Universal Robots URScript: pick_up_bottle_cups_xijun.script

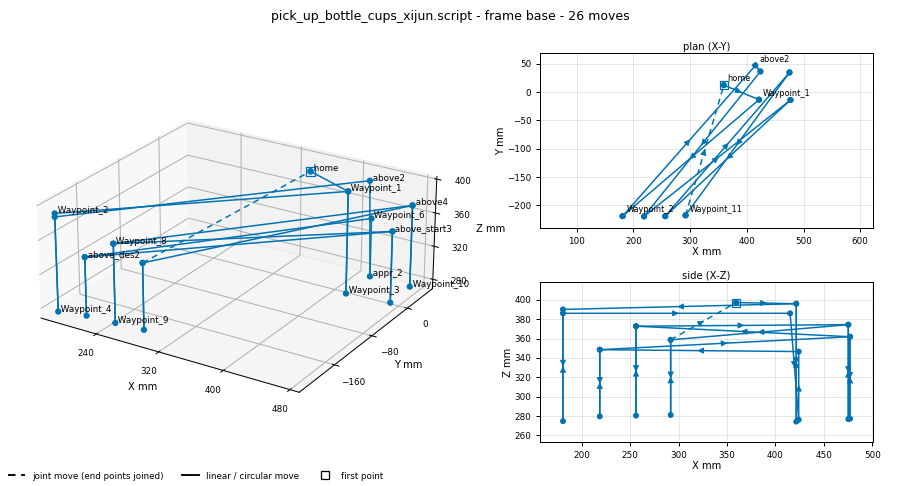
[picture p0: tool path of pick_up_bottle_cups_xijun.script in frame base, 26 of 27 moves have a stored position in this frame; points joined in program order, loops and branches not executed]
def pick_up_bottle_cups_xijun():
  set_tool_communication(True, 1000000, 2, 1, 1.5, 3.5)
  set_tool_output_mode(0)
  set_tool_digital_output_mode(0, 1)
  set_tool_digital_output_mode(1, 1)
  set_tool_voltage(24)
  set_tcp(p[0.0,0.0,0.0,0.0,0.0,0.0])
  set_target_payload(1.070000, [0.002000, 0.003000, 0.057000], [0.001723, 0.001723, 0.001723, 0.000000, 0.000000, 0.000000])
  set_safety_mode_transition_hardness(1)
  set_standard_analog_input_domain(0, 1)
  set_standard_analog_input_domain(1, 1)
  set_tool_analog_input_domain(0, 1)
  set_tool_analog_input_domain(1, 1)
  set_analog_outputdomain(0, 0)
  set_analog_outputdomain(1, 0)
  set_input_actions_to_default()
  step_count_40e01536_ad7e_4052_bcf8_2e85b5cb6fec = 0.0
  thread Step_Counter_Thread_e9fd1985_c531_4e2b_8333_d58f243b9e86():
    while (True):
      step_count_40e01536_ad7e_4052_bcf8_2e85b5cb6fec = step_count_40e01536_ad7e_4052_bcf8_2e85b5cb6fec + 1.0
      sync()
    end
  end
  run Step_Counter_Thread_e9fd1985_c531_4e2b_8333_d58f243b9e86()
  set_gravity([0.0, 0.0, 9.82])
  global Pallet_3_cnt=1
  global Plane_1=p[-0.700006141123905,1.3454883874109249E-6,0.3910559577028425,-1.2089868272251132,-1.2089999932245832,1.20858562628424]
  global Plane_2=p[0.0,0.0,0.0,0.0,0.0,0.0]
  global Point_1=p[0.6913645118948067,-0.12399382748223003,0.49223711947071,-1.2983729986843258,1.1259514972191385,-1.2203503861141718]
  # begin: URCap Installation Node
  #   Source: External Control, 1.0.5, FZI Research Center for Information Technology
  #   Type: External Control
  # end: URCap Installation Node
  # begin: URCap Installation Node
  #   Source: OnRobot, 6.2.0, OnRobot A/S
  #   Type: OnRobot Setup
  sleep(1)
  if (False):
    global rg_Busy = 0
    global rg_Depth = 0
    global rg_DepthRel = 0
    global rg_Grip_detected = 0
    global rg_Width = 0
  end
  ON_CONN_SHIFT_BOOL = 64
  ON_CONN_SHIFT_INT = 24
  ON_CONN_SHIFT_FLOAT = 24
  ON_CONN_REG_SUM_BOOL = 7
  ON_CONN_REG_SUM_INT = 4
  ON_CONN_REG_SUM_FLOAT = 3
  ON_TOOL_SHIFT_BOOL = 64
  ON_TOOL_SHIFT_INT = 25
  ON_TOOL_SHIFT_FLOAT = 24
  ON_TOOL_SHIFT_BOOL_ARR = [64, 71, 71]
  ON_TOOL_SHIFT_INT_ARR = [25, 28, 28]
  ON_TOOL_SHIFT_FLOAT_ARR = [24, 27, 27]
  ON_TOOL_REG_SUM_BOOL = 7
  ON_TOOL_REG_SUM_INT = 3
  ON_TOOL_REG_SUM_FLOAT = 3
  ON_REGISTERS_SPEEDL_FLOAT = 0
  ON_REG_USE_TOOL = False
  ON_DI_SINGLE = 0
  ON_DI_PRIMARY = 1
  ON_DI_SECONDARY = 2
  ON_DI_DUAL = 3
  on_robot_type = 10
  on_robot_cycle = 2.0
  on_conn_ip = "localhost"
  on_tool_ip = "localhost"
  on_device_socket_port = 51234
  on_conn_xmlrpc = rpc_factory("xmlrpc", "http://localhost:41414")
  on_tool_xmlrpc = rpc_factory("xmlrpc", "http://localhost:41414")
  on_RPC = rpc_factory("xmlrpc", "http://127.0.0.1:31416")
  ON_DEBUG_LOG = False
  on_isMetric = True
  on_toolConnector = True
  on_ioqc = False
  on_dual = False
  on_computebox = False
  on_devices = 1
  on_gripper = [False, False, False]
  on_custom_tcp_id = "none"
  on_custom_tcp_enabled = False
  speedlTime = 0.001
  on_ft = False
  rg_index = 0
  on_gripper[rg_index] = True
  #======    OnRobot Globals    ======#

  ON_MATH_PI=3.141593
  ON_ZEROPOSE=p[0.0,0.0,0.0,0.0,0.0,0.0]
  ON_ZEROFRAME=p[0.0,0.0,0.0,0.0,0.0,0.0]
  ON_ZERO3D=[0.0,0.0,0.0]
  ON_ZERO6D=[0.0,0.0,0.0,0.0,0.0,0.0]
  ON_ZERO8D=[0.0,0.0,0.0,0.0,0.0,0.0,0.0,0.0]
  ON_FALSE3D=[False,False,False]
  ON_FALSE6D=[False,False,False,False,False,False]
  ON_FALSE8D=[False,False,False,False,False,False,False,False]
  global on_return=0
  on_speedL=ON_ZERO6D
  on_speedBase=ON_ZERO6D
  on_speedVect=ON_ZERO6D
  on_speedExtra=ON_ZERO6D
  on_speedCB=ON_ZERO6D
  on_speedGecko=ON_ZERO6D
  on_RTDE_error=0
  on_RTDE_tool_error=0
  on_dataProcess_thrd=0
  ON_DEVICE_ID_MISSING=0
  ON_INIT_WATCHDOG_HZ=5
  ON_INIT_TIMEOUT=2000
  on_robot_TCP_offset=ON_ZEROFRAME
  on_tcp_offset_actual=ON_ZEROFRAME
  on_cog_actual=ON_ZEROFRAME
  on_mass_actual=0.0
  on_robot_mount=[0.0,0.0]

  #======    End of OnRobot Globals    ======#
  #======    OnRobot RG Globals    ======#

  RG_DEVICE_ID_RG2=32
  RG_DEVICE_ID_RG6=33
  if ON_DEBUG_LOG:
  textmsg("RG Dual: False, Index: ",rg_index)
  if False:
  rg_index=-1
  end
  end
  rg_Width_arr=[0,0,0]
  rg_Depth_arr=[0,0,0]
  rg_DepthRel_arr=[0,0,0]
  rg_product_code_arr=[0,0,0]
  rg_device_id_arr=[0,0,0]
  rg_Status_arr=[0,0,0]
  rg_Grip_detected_arr=[False,False,False]
  rg_Busy_arr=[False,False,False]
  rg_S1_pushed_arr=[False,False,False]
  rg_S1_triggered_arr=[False,False,False]
  rg_S2_pushed_arr=[False,False,False]
  rg_S2_triggered_arr=[False,False,False]
  rg_Safety_error_arr=[False,False,False]
  rg_Speed_arr=[0,0,0]
  rg_Angle_arr=[0,0,0]
  rg_Angle_speed_arr=[0,0,0]
  rg_Depth_prev_arr=[0,0,0]
  rg_speedDC=ON_ZERO6D
  rg_data_error_arr=[0,0,0]
  rg_mounting_angle_arr=[0,0,0]
  rg_fingertip_arr=[0,0,0]
  rg_Grip_guard_arr=[False,False,False]

  rg_Width=0
  rg_Depth=0
  rg_DepthRel=0
  rg_Busy=False
  rg_Grip_detected=False
  def get_rg_Width():
  return rg_Width
  end
  def get_rg_Depth():
  return rg_Depth
  end
  def get_rg_DepthRel():
  return rg_DepthRel
  end
  def get_rg_Busy():
  return rg_Busy
  end
  def get_rg_Grip_detected():
  return rg_Grip_detected
  end

  rg2_mount_bracket_offset=35.0/1000.0
  rg2_mount_body_offset=p[0.0,0.0,0.180,0.0,0.0,0.0]
  rg2_mount_cog_offset=p[0.0,0.0,0.065,0.0,0.0,0.0]
  rg6_mount_bracket_offset=35.0/1000.0
  rg6_mount_body_offset=p[0.0,0.0,0.230,0.0,0.0,0.0]
  rg6_mount_cog_offset=p[0.0,0.0,0.080,0.0,0.0,0.0]

  #======    End of OnRobot RG Globals    ======#
  #======    OnRobot Interface Messages    ======#

  on_devices_primary_log="OnRobot Devices"
  on_devices_secondary_log="OnRobot Secondary Device"
  on_program_halted="<br>Program halted."
  on_device_error_title="OnRobot - Device error"
  on_install_error="OnRobot Setup is not correct.<br>Check the status in the OnRobot Setup page in the Installation Tab.<br>Program halted."
  on_device_missing="No device connected.<br>Program halted."
  cb_device_missing="No OnRobot Compute Box connected.<br>Program halted."
  ft_device_missing="No OnRobot FT sensor or license detected.<br>Program halted."
  hex_device_missing="No HEX sensor connected.<br>Program halted."
  rg2ft_device_missing="No RG2-FT gripper connected.<br>Program halted."
  rg_device_missing="No RG gripper connected.<br>Program halted."
  vg_device_missing="No VG gripper connected.<br>Program halted."
  gg_device_missing="No Gecko Gripper connected.<br>Program halted."
  sg_device_missing="No Soft Gripper connected.<br>Program halted."
  tfg_device_missing="No 3FG gripper connected.<br>Program halted."
  sdr_device_missing="No OnRobot Sander connected.<br>Program halted."
  twofg_device_missing="No 2FG gripper connected.<br>Program halted."
  vgp_device_missing="No VGP gripper connected.<br>Program halted."
  mg_device_missing="No Magnetic Gripper connected.<br>Program halted."
  fgp_device_missing="No 2FGP20 Gripper connected.<br>Program halted."
  eyes_device_missing="No OnRobot Eyes connected.<br>Program halted."
  on_xmlrpc_start_ip="Connecting to OnRobot XML-RPC Server:"
  on_java_comm_error_textmsg_title="OnRobot - Communication error:"
  on_java_comm_controlsocket_open_error="Socket 'javaSocket' opening was unsuccessful."
  on_java_comm_error_title="OnRobot - Communication error"
  on_java_comm_socket_open_error="Establishing connection with the URCap was timed out.<br>Check the status in the OnRobot Setup page in the Installation Tab.<br>Program halted."
  on_rtde_feed_error_textmsg_title="OnRobot - RTDE error:"
  on_rtde_feed_error="RTDE feed error. OnRobot device count mismatch.<br>Program halted."
  on_rtde_feed_tool_error="Tool RTDE feed error. OnRobot device count mismatch.<br>Program halted."
  on_rtde_feed_open_error_textmsg="Socket 'rtdeFeed' opening was unsuccessful."
  on_rtde_feed_error_title="OnRobot - RTDE error"
  on_rtde_feed_count_error="Invalid RTDE offset setup detected. Please check RTDE Offsets at the OnRobot Setup page in the Installation Tab.<br>Program halted."
  on_rtde_feed_open_error="Establishing connection with the devices was timed out.<br>Ensure that the OnRobot devices are operational, and check the status in the OnRobot Setup page in the Installation Tab."

  #======    End of OnRobot Interface Messages    ======#
  #======    OnRobot Interface    ======#

  on_portopened_javaSocket=False
  on_rtde_feed_opened=False
  on_dataProcess_running=False
  def on_missing():
  popup(on_device_missing,title=on_device_error_title,error=True,blocking=False)
  halt
  end
  def cb_missing():
  popup(cb_device_missing,title=on_device_error_title,error=True,blocking=False)
  halt
  end
  def ft_missing():
  popup(ft_device_missing,title=on_device_error_title,error=True,blocking=False)
  halt
  end
  def hex_missing():
  popup(hex_device_missing,title=on_device_error_title,error=True,blocking=False)
  halt
  end
  def rg2ft_missing():
  popup(rg2ft_device_missing,title=on_device_error_title,error=True,blocking=False)
  halt
  end
  def rg_missing():
  popup(rg_device_missing,title=on_device_error_title,error=True,blocking=False)
  halt
  end
  def vg_missing():
  popup(vg_device_missing,title=on_device_error_title,error=True,blocking=False)
  halt
  end
  def gg_missing():
  popup(gg_device_missing,title=on_device_error_title,error=True,blocking=False)
  halt
  end
  def sg_missing():
  popup(sg_device_missing,title=on_device_error_title,error=True,blocking=False)
  halt
  end
  def tfg_missing():
  popup(tfg_device_missing,title=on_device_error_title,error=True,blocking=False)
  halt
  end
  def sdr_missing():
  popup(sdr_device_missing,title=on_device_error_title,error=True,blocking=False)
  halt
  end
  def twofg_missing():
  popup(twofg_device_missing,title=on_device_error_title,error=True,blocking=False)
  halt
  end
  def vgp_missing():
  popup(vgp_device_missing,title=on_device_error_title,error=True,blocking=False)
  halt
  end
  def mg_missing():
  popup(mg_device_missing,title=on_device_error_title,error=True,blocking=False)
  halt
  end
  def fgp_missing():
  popup(fgp_device_missing,title=on_device_error_title,error=True,blocking=False)
  halt
  end
  def eyes_missing():
  popup(eyes_device_missing,title=on_device_error_title,error=True,blocking=False)
  halt
  end
  def on_portclose_javaSocket():
  socket_close("javaSocket")
  on_portopened_javaSocket=False
  end
  def on_portopen_javaSocket():
  on_portclose_javaSocket()
  on_portopened_javaSocket=socket_open("127.0.0.1",44005,"javaSocket")
  if not on_portopened_javaSocket:
  textmsg(on_java_comm_error_textmsg_title,on_java_comm_controlsocket_open_error)
  popup(on_java_comm_socket_open_error,title=on_java_comm_error_title,error=True,blocking=False)
  halt
  end
  end
  on_conn_rtde_feed_name="rtdeFeedConn"
  on_tool_rtde_feed_name="rtdeFeedTool"
  def on_rtde_feed_close(rtdeFeedName):
  socket_close(rtdeFeedName)
  on_rtde_feed_opened=False
  end
  def on_rtde_feed_open(deviceIP,rtdeFeedName,regStart,regSum,regSpeedl):
  on_rtde_feed_close(rtdeFeedName)
  if((regStart[0]+regSum[0])>128)or((regStart[1]+regSum[1])>48)or((regStart[2]+regSum[2])>48):
  popup(on_rtde_feed_count_error,title=on_rtde_feed_error_title,error=True,blocking=False)
  textmsg(str_cat("RegStart: ",regStart),str_cat("  -  RegSum: ",regSum))
  halt
  end
  on_rtde_feed_opened=socket_open(deviceIP,on_device_socket_port,rtdeFeedName)
  if not on_rtde_feed_opened:
  on_rtde_feed_opened=socket_open(deviceIP,on_device_socket_port,rtdeFeedName)
  end
  if not on_rtde_feed_opened:
  textmsg(on_rtde_feed_error_textmsg_title,on_rtde_feed_open_error_textmsg)
  popup(on_rtde_feed_open_error,title=on_rtde_feed_error_title,error=True,blocking=False)
  halt
  end
  socket_send_int(regStart[0],rtdeFeedName)
  socket_send_int(regSum[0],rtdeFeedName)
  socket_send_int(regStart[1],rtdeFeedName)
  socket_send_int(regSum[1],rtdeFeedName)
  socket_send_int(regStart[2],rtdeFeedName)
  socket_send_int(regSum[2],rtdeFeedName)
  socket_send_int(regSpeedl,rtdeFeedName)
  socket_send_int(on_devices,rtdeFeedName)
  end
  def on_dataRead():
  enter_critical
  on_RTDE_error=read_input_integer_register(ON_CONN_SHIFT_INT)
  if(ON_REG_USE_TOOL):
  on_RTDE_tool_error=read_input_integer_register(ON_TOOL_SHIFT_INT_ARR[0])
  end
  exit_critical
  end
  def on_set_rtde_watchdog(updateHz=ON_INIT_WATCHDOG_HZ):
  local effect="stop"
  if(updateHz<1):
  effect="ignore"
  end
  watchdog_conn_reg_str=str_cat("input_int_register_",ON_CONN_SHIFT_INT)
  rtde_set_watchdog(watchdog_conn_reg_str,updateHz,effect)
  if(ON_REG_USE_TOOL):
  watchdog_tool_reg_str=str_cat("input_int_register_",ON_TOOL_SHIFT_INT_ARR[0])
  rtde_set_watchdog(watchdog_tool_reg_str,updateHz,effect)
  end
  if ON_DEBUG_LOG:
  local update_str=str_cat(" "+effect+" watchdog set to [Hz]: ",updateHz)
  textmsg(watchdog_conn_reg_str,update_str)
  if(ON_REG_USE_TOOL):
  local update_str=str_cat(" "+effect+" watchdog set to [Hz]: ",updateHz)
  textmsg(watchdog_tool_reg_str,update_str)
  end
  end
  end
  def on_speedCB_get():
  return[on_speedCB[0],on_speedCB[1],on_speedCB[2],on_speedCB[3],on_speedCB[4],on_speedCB[5]]
  end
  def on_speedGecko_get():
  local speedExtra=ON_ZERO6D
  if on_speedl_for_gecko:
  speedExtra=[on_speedGecko[0],on_speedGecko[1],on_speedGecko[2],on_speedGecko[3],on_speedGecko[4],on_speedGecko[5]]
  end
  return speedExtra
  end
  def on_speedGecko_set(speedGecko):
  on_speedGecko=[speedGecko[0],speedGecko[1],speedGecko[2],speedGecko[3],speedGecko[4],speedGecko[5]]
  end
  thread on_dataProcess_thread():
  if ON_DEBUG_LOG:
  textmsg("Starting on_dataRead thread")
  end
  local error=False
  on_dataProcess_running=True
  sync()
  while on_dataProcess_running:
  sync()
  on_dataRead()
  error=on_error((on_RTDE_error<0),on_rtde_feed_error,on_rtde_feed_error_title,error)
  error=on_error((ON_REG_USE_TOOL and(on_RTDE_tool_error<0)),on_rtde_feed_tool_error,on_rtde_feed_error_title,error)
  on_dataProcess_running=not error
  end
  if error:
  halt
  end
  if ON_DEBUG_LOG:
  textmsg("Stopping on_dataRead thread")
  end
  end
  thread on_set_watchdog_thread():
  sleep(2)
  on_set_rtde_watchdog(updateHz=ON_INIT_WATCHDOG_HZ)
  sleep(1/ON_INIT_WATCHDOG_HZ)
  on_dataProcess_running=False
  kill on_dataProcess_thrd
  end

  #======    End of OnRobot Interface    ======#
  #======    OnRobot QC Setup Tool Connector    ======#

  def tc_setup_tool():
  if ON_DEBUG_LOG:
  textmsg("QC Setup Tool Connector start...")
  end
  set_tool_voltage(24)

  set_tool_communication(True,1000000,2,1,1.5,3.5)

  if ON_DEBUG_LOG:
  textmsg("QC Setup Tool Connector end.")
  end
  end

  #======    End of OnRobot QC Setup Tool Connector    ======#
  #======    OnRobot RG Interface    ======#

  rg_dataRead_running=False
  def rg_dataRead_RTDE(tool_index):
  local reg_offset_bool=ON_TOOL_SHIFT_BOOL_ARR[tool_index]
  local reg_offset_int=ON_TOOL_SHIFT_INT_ARR[tool_index]
  local reg_offset_float=ON_TOOL_SHIFT_FLOAT_ARR[tool_index]
  enter_critical
  floatRegDummy=read_input_float_register(reg_offset_float+0)
  rg_Width_arr[tool_index]=floatRegDummy
  floatRegDummy=read_input_float_register(reg_offset_float+1)
  rg_Depth_arr[tool_index]=floatRegDummy
  floatRegDummy=read_input_float_register(reg_offset_float+2)
  rg_DepthRel_arr[tool_index]=floatRegDummy
  intRegDummy=read_input_integer_register(reg_offset_int+0)
  rg_device_id_arr[tool_index]=intRegDummy
  intRegDummy=read_input_integer_register(reg_offset_int+1)
  rg_product_code_arr[tool_index]=intRegDummy
  intRegDummy=read_input_integer_register(reg_offset_int+2)
  rg_Status_arr[tool_index]=intRegDummy
  boolRegDummy=read_input_boolean_register(reg_offset_bool+0)
  rg_Busy_arr[tool_index]=boolRegDummy
  boolRegDummy=read_input_boolean_register(reg_offset_bool+1)
  rg_Grip_detected_arr[tool_index]=boolRegDummy
  boolRegDummy=read_input_boolean_register(reg_offset_bool+2)
  rg_S1_pushed_arr[tool_index]=boolRegDummy
  boolRegDummy=read_input_boolean_register(reg_offset_bool+3)
  rg_S1_triggered_arr[tool_index]=boolRegDummy
  boolRegDummy=read_input_boolean_register(reg_offset_bool+4)
  rg_S2_pushed_arr[tool_index]=boolRegDummy
  boolRegDummy=read_input_boolean_register(reg_offset_bool+5)
  rg_S2_triggered_arr[tool_index]=boolRegDummy
  boolRegDummy=read_input_boolean_register(reg_offset_bool+6)
  rg_Safety_error_arr[tool_index]=boolRegDummy
  exit_critical
  end
  thread rg_dataRead_thread():
  if ON_DEBUG_LOG:
  textmsg("Starting rg_dataRead thread")
  end
  while rg_dataRead_running:
  sync()
  rg_Depth_prev_arr=rg_Depth_arr
  if(rg_index==ON_DI_DUAL):
  rg_dataRead_RTDE(ON_DI_PRIMARY)
  rg_dataRead_RTDE(ON_DI_SECONDARY)
  else:
  rg_dataRead_RTDE(rg_index)
  end
  end
  if ON_DEBUG_LOG:
  textmsg("Stopping rg_dataRead thread")
  end
  end

  #======    End of OnRobot RG Interface    ======#
  #======    OnRobot TCP Messages    ======#

  on_tcp_log_msg_default="OnRobot: Robot TCP Offset set to:"
  on_tcp_log_msg_primary="OnRobot: Robot TCP Offset set to Primary:"
  on_tcp_log_msg_secondary="OnRobot: Robot TCP Offset set to Secondary:"

  #======    End of OnRobot TCP Messages    ======#
  #======    OnRobot TCP    ======#

  on_tcp_offset_actual=ON_ZEROFRAME
  on_tcp_offset_primary=ON_ZEROFRAME
  on_tcp_static_primary=ON_ZEROFRAME
  on_tcp_dynamic_primary=ON_ZEROFRAME
  on_tcp_adapters=ON_ZEROFRAME
  on_tcp_qc_primary=ON_ZEROFRAME
  on_tcp_base_primary=ON_ZEROFRAME
  on_tcp_gripper_static_primary=ON_ZEROFRAME
  on_tcp_workpiece_primary=ON_ZEROFRAME
  on_tcp_gripper_dynamic_primary=ON_ZEROFRAME
  on_tcp_gripper_primary=ON_ZEROFRAME
  on_tcp_offset_secondary=ON_ZEROFRAME
  on_tcp_static_secondary=ON_ZEROFRAME
  on_tcp_dynamic_secondary=ON_ZEROFRAME
  on_tcp_qc_secondary=ON_ZEROFRAME
  on_tcp_base_secondary=ON_ZEROFRAME
  on_tcp_gripper_static_secondary=ON_ZEROFRAME
  on_tcp_workpiece_secondary=ON_ZEROFRAME
  on_tcp_gripper_dynamic_secondary=ON_ZEROFRAME
  on_tcp_gripper_secondary=ON_ZEROFRAME
  on_tcp_custom_preset_assigned=False
  on_tcp_custom_preset=ON_ZEROFRAME
  def on_tcp_init_adapters():
  if ON_DEBUG_LOG:
  textmsg("TCP Init Adapters start..")
  end
  enter_critical
  on_tcp_adapters=ON_ZEROFRAME
  local adapterCount=length(on_tcp_adapters_array)
  local i=0
  while(i<adapterCount):
  on_tcp_adapters=pose_trans(on_tcp_adapters,on_tcp_adapters_array[i])
  i=i+1
  end
  exit_critical
  if ON_DEBUG_LOG:
  textmsg("TCP Init Adapters end.")
  end
  end
  def on_tcp_update_primary():
  if ON_DEBUG_LOG:
  textmsg("TCP Update Primary start..")
  end
  on_tcp_gripper_dynamic_primary=p[0.0, 0.0, 0.0, 0.0, 0.0, 0.0]
  enter_critical
  on_tcp_dynamic_primary=pose_trans(on_tcp_static_primary,on_tcp_gripper_dynamic_primary)
  on_tcp_offset_primary=pose_trans(on_tcp_dynamic_primary,on_tcp_workpiece_primary)
  exit_critical
  if ON_DEBUG_LOG:
  textmsg("TCP Update Primary end.")
  end
  end
  def on_tcp_init_primary():
  if ON_DEBUG_LOG:
  textmsg("TCP Init Primary start..")
  end
  enter_critical
  on_tcp_base_primary=pose_trans(on_tcp_adapters,on_tcp_qc_primary)
  on_tcp_static_primary=pose_trans(on_tcp_base_primary,on_tcp_gripper_static_primary)
  exit_critical
  on_tcp_update_primary()
  if ON_DEBUG_LOG:
  textmsg("TCP Init Primary end.")
  end
  end
  def on_tcp_offset_set(TCP_offset):
  if ON_DEBUG_LOG:
  textmsg("TCP Offset set started!")
  end
  on_tcp_offset_send(TCP_offset)
  if(on_follow_tcp):
  set_tcp(TCP_offset)
  end
  on_robot_TCP_offset=TCP_offset
  if ON_DEBUG_LOG:
  textmsg("TCP Offset set to: ",on_robot_TCP_offset)
  end
  end
  def on_tcp_offset_forced_set_actual(isPrimary=True):
  if(not on_follow_tcp):

  local tcp_log_msg=on_tcp_log_msg_default

  textmsg(tcp_log_msg,on_tcp_offset_actual)
  set_tcp(on_tcp_offset_actual)
  end
  end
  def on_tcp_update(isPrimary=True):
  on_tcp_update_primary()

  on_tcp_set_actual_to(isPrimary)
  end
  def on_tcp_set_actual_to(isPrimary=True):

  on_tcp_offset_actual=on_tcp_offset_primary
  if(on_follow_tcp):
  textmsg(on_tcp_log_msg_default,on_tcp_offset_actual)
  end

  on_tcp_active_is_primary=isPrimary
  on_tcp_offset_set(on_tcp_offset_actual)
  end
  def on_tcp_update_workpiece_primary(workpiece_offset):
  if ON_DEBUG_LOG:
  textmsg("TCP Update Tool Primary start..")
  end
  on_tcp_workpiece_primary=workpiece_offset
  on_tcp_update_primary()
  if ON_DEBUG_LOG:
  textmsg("TCP Update Tool Primary end.")
  end
  end
  def on_tcp_workpiece_rpy_get(xyz=[0.0,0.0,0.0],rpy=[0.0,0.0,0.0]):
  local rotvec=rpy2rotvec(rpy)
  local workpiece_offset=p[xyz[0],xyz[1],xyz[2],rotvec[0],rotvec[1],rotvec[2]]
  return workpiece_offset
  end

  def on_tcp_update_workpiece(workpiece_offset,tool_index=0):
  if ON_DEBUG_LOG:
  textmsg("TCP Update Tool start..")
  end
  if(tool_index!=ON_DI_SECONDARY):
  on_tcp_update_workpiece_primary(workpiece_offset)
  local isPrimary=True

  end
  on_tcp_set_actual_to(isPrimary)
  if ON_DEBUG_LOG:
  textmsg("TCP Update Tool end.")
  end
  end
  def on_get_tcp_for(tool_index):
  if tool_index==ON_DI_SECONDARY:
  local actual_tcp=on_tcp_static_secondary
  else:
  local actual_tcp=on_tcp_static_primary
  end
  return actual_tcp
  end
  def on_tcp_custom_unused():
  return ON_ZEROFRAME
  end
  def on_tcp_update_custom():
  if ON_DEBUG_LOG:
  textmsg("TCP Update Custom start..")
  end
  if(on_custom_tcp_enabled):
  on_tcp_custom_unused()
  on_tcp_custom_unused()
  on_tcp_custom_unused()
  on_tcp_custom_unused()

  end
  if ON_DEBUG_LOG:
  textmsg("TCP Update Custom end.")
  end
  end

  #======    End of OnRobot TCP    ======#
  #======    OnRobot Payload Messages    ======#

  on_mass_log_msg="OnRobot: Robot Payload Mass set to:"
  on_cog_log_msg="OnRobot: Robot Payload Center of Gravity set to:"

  #======    End of OnRobot Payload Messages    ======#
  #======    OnRobot Payload    ======#

  on_cog_actual=ON_ZEROFRAME
  on_mass_actual=0.0
  on_cog_primary=ON_ZEROFRAME
  on_cog_L1L2_primary=ON_ZEROFRAME
  on_mass_primary=0.0
  on_mass_L1L2_primary=0.0
  on_cog_adapters=ON_ZEROFRAME
  on_cog_qc_primary=ON_ZEROFRAME
  on_cog_base_primary=ON_ZEROFRAME
  on_cog_gripper_primary=ON_ZEROFRAME
  on_cog_workpiece_primary=ON_ZEROFRAME
  on_mass_adapters=0.0
  on_mass_qc_primary=0.0
  on_mass_base_primary=0.0
  on_mass_gripper_primary=0.0
  on_mass_workpiece_primary=0.0
  on_cog_secondary=ON_ZEROFRAME
  on_mass_secondary=0.0
  on_cog_gripper_secondary=ON_ZEROFRAME
  on_mass_gripper_secondary=0.0
  on_cog_workpiece_secondary=ON_ZEROFRAME
  on_mass_workpiece_secondary=0.0
  ON_LB2KG001=0.45359237/100
  def on_payload_init_adapters():
  if ON_DEBUG_LOG:
  textmsg("TCP Init Adapters start..")
  end
  enter_critical
  on_cog_adapters=ON_ZEROFRAME
  on_mass_adapters=0.0
  local massLAL0Ratio=0
  local adapterAbsCOG=ON_ZEROFRAME
  local tcp_adapter_offset=ON_ZEROFRAME
  local adapterCount=length(on_tcp_adapters_array)
  local i=0
  while(i<adapterCount):
  on_mass_adapters=on_mass_adapters+on_mass_adapters_array[i]
  if(on_mass_adapters<=0):
  massLAL0Ratio=0
  else:
  massLAL0Ratio=on_mass_adapters_array[i]/on_mass_adapters
  end
  adapterAbsCOG=pose_trans(tcp_adapter_offset,on_tcp_adapters_array[i])
  adapterAbsCOG=p[adapterAbsCOG[0],adapterAbsCOG[1],adapterAbsCOG[2],0.0,0.0,0.0]
  on_cog_adapters=interpolate_pose(on_cog_adapters,adapterAbsCOG,massLAL0Ratio)
  on_cog_adapters=p[on_cog_adapters[0],on_cog_adapters[1],on_cog_adapters[2],0.0,0.0,0.0]
  tcp_adapter_offset=pose_trans(tcp_adapter_offset,on_tcp_adapters_array[i])
  i=i+1
  sync()
  end
  exit_critical
  if ON_DEBUG_LOG:
  textmsg("TCP Init Adapters end.")
  end
  end
  def on_payload_update_primary():
  if ON_DEBUG_LOG:
  textmsg("Payload Update Primary start..")
  end
  enter_critical
  on_mass_primary=on_mass_L1L2_primary+on_mass_workpiece_primary
  local massL1L2L3Ratio=on_mass_workpiece_primary/on_mass_primary
  local workpieceAbsCOG=pose_trans(on_tcp_dynamic_primary,on_cog_workpiece_primary)
  workpieceAbsCOG=p[workpieceAbsCOG[0],workpieceAbsCOG[1],workpieceAbsCOG[2],0.0,0.0,0.0]
  on_cog_primary=interpolate_pose(on_cog_L1L2_primary,workpieceAbsCOG,massL1L2L3Ratio)
  on_cog_primary=p[on_cog_primary[0],on_cog_primary[1],on_cog_primary[2],0.0,0.0,0.0]
  exit_critical
  if ON_DEBUG_LOG:
  textmsg("Payload Update Primary end.")
  end
  end
  def on_payload_init_primary():
  if ON_DEBUG_LOG:
  textmsg("Payload Init Primary start..")
  end
  enter_critical
  on_mass_base_primary=on_mass_adapters+on_mass_qc_primary
  local massL0L1Ratio=on_mass_qc_primary/on_mass_base_primary
  on_mass_L1L2_primary=on_mass_base_primary+on_mass_gripper_primary
  local massL1L2Ratio=on_mass_gripper_primary/on_mass_L1L2_primary
  local qcAbsCOG=pose_trans(on_tcp_adapters,on_cog_qc_primary)
  qcAbsCOG=p[qcAbsCOG[0],qcAbsCOG[1],qcAbsCOG[2],0.0,0.0,0.0]
  on_cog_base_primary=interpolate_pose(on_cog_adapters,qcAbsCOG,massL0L1Ratio)
  on_cog_base_primary=p[on_cog_base_primary[0],on_cog_base_primary[1],on_cog_base_primary[2],0.0,0.0,0.0]
  local gripperAbsCOG=pose_trans(on_tcp_base_primary,on_cog_gripper_primary)
  gripperAbsCOG=p[gripperAbsCOG[0],gripperAbsCOG[1],gripperAbsCOG[2],0.0,0.0,0.0]
  on_cog_L1L2_primary=interpolate_pose(on_cog_base_primary,gripperAbsCOG,massL1L2Ratio)
  on_cog_L1L2_primary=p[on_cog_L1L2_primary[0],on_cog_L1L2_primary[1],on_cog_L1L2_primary[2],0.0,0.0,0.0]
  exit_critical
  on_payload_update_primary()
  if ON_DEBUG_LOG:
  textmsg("Payload Init Primary end.")
  end
  end
  def on_payload_update():
  on_payload_update_primary()

  on_mass_actual =on_mass_primary
  on_cog_actual=on_cog_primary

  on_payload_set_actual()
  end
  def on_payload_set_actual():

  on_mass_actual =on_mass_primary
  on_cog_actual=on_cog_primary

  local CoG=[on_cog_actual[0],on_cog_actual[1],on_cog_actual[2]]
  on_payload_set(on_mass_actual,CoG)
  end
  def on_payload_update_workpiece_primary(workpiece_mass=0,workpiece_cog=[0.0,0.0,0.0]):
  if ON_DEBUG_LOG:
  textmsg("Payload Update Workpiece Primary start..")
  end
  on_cog_workpiece_primary=p[workpiece_cog[0],workpiece_cog[1],workpiece_cog[2],0.0,0.0,0.0]
  on_mass_workpiece_primary=workpiece_mass
  on_payload_update_primary()
  if ON_DEBUG_LOG:
  textmsg("Payload Update Workpiece Primary end.")
  end
  end
  def on_payload_set(mass,CoG):
  if ON_DEBUG_LOG:
  textmsg("Payload set started!")
  end
  local center_of_gravity=[CoG[0],CoG[1],CoG[2]]
  on_payload_send(center_of_gravity,mass)
  if(on_isMetric):
  local roundedMass=floor(mass*100+0.5)/100
  else:
  local roundedMass=floor(mass/ON_LB2KG001+0.5)*ON_LB2KG001
  end
  set_payload(roundedMass,center_of_gravity)
  on_mass_actual=roundedMass
  on_cog_actual=p[CoG[0],CoG[1],CoG[2],0.0,0.0,0.0]
  if ON_DEBUG_LOG:
  textmsg("Payload mass, CoG set to: ",str_cat(str_cat(mass,", "),CoG))
  end
  end

  def on_payload_update_secondary():
  end
  def on_payload_init_secondary():
  end

  def on_payload_update_workpiece(workpiece_mass,workpiece_cog=[0.0,0.0,0.0],tool_index=0):
  if ON_DEBUG_LOG:
  textmsg("Payload Update Workpiece start..")
  end
  if(tool_index!=ON_DI_SECONDARY):
  on_cog_workpiece_primary=p[workpiece_cog[0],workpiece_cog[1],workpiece_cog[2],0.0,0.0,0.0]
  on_mass_workpiece_primary=workpiece_mass
  else:
  on_cog_workpiece_secondary=p[workpiece_cog[0],workpiece_cog[1],workpiece_cog[2],0.0,0.0,0.0]
  on_mass_workpiece_secondary=workpiece_mass
  end
  on_payload_update()
  if ON_DEBUG_LOG:
  textmsg("Payload Update Workpiece end.")
  end
  end
  def on_payload_get_cog2tcp_workpiece(tool_index=0):
  if(tool_index!=ON_DI_SECONDARY):
  local cog_tool=[on_tcp_workpiece_primary[0],on_tcp_workpiece_primary[1],on_tcp_workpiece_primary[2]]
  else:
  local cog_tool=[on_tcp_workpiece_secondary[0],on_tcp_workpiece_secondary[1],on_tcp_workpiece_secondary[2]]
  end
  return cog_tool
  end

  #======    End of OnRobot Payload    ======#
  #======    OnRobot QC TCP    ======#

  onrobotmini=0

  def on_tcp_offset_send(TCP_offset):
  on_robot_TCP_offset=TCP_offset
  end
  def on_payload_send(CoG,mass):
  on_robot_payload_cog=CoG
  on_robot_payload_mass=mass
  end


  #======    End of OnRobot QC TCP    ======#
  #======    OnRobot RG TCP    ======#

  def rg_mount_tcp(gripper_angle,isRG2=True):
  if ON_DEBUG_LOG:
  textmsg("RG Mount TCP command starting..")
  end
  if(isRG2):
  local gripperBracket=rg2_mount_bracket_offset
  local gripperBody=rg2_mount_body_offset
  else:
  local gripperBracket=rg6_mount_bracket_offset
  local gripperBody=rg6_mount_body_offset
  end
  local gripperRotVec=rpy2rotvec([gripper_angle,0.0,0.0])
  local gripperMountOffset=p[0.0,0.0,gripperBracket,gripperRotVec[0],gripperRotVec[1],gripperRotVec[2]]
  local gripperOffsetStatic=pose_trans(gripperMountOffset,gripperBody)
  if ON_DEBUG_LOG:
  textmsg("RG Mount TCP command ended.")
  end
  return gripperOffsetStatic
  end
  def rg_mount_cog(gripper_angle,isRG2=True):
  if ON_DEBUG_LOG:
  textmsg("RG Mount CoG command starting..")
  end
  if(isRG2):
  local gripperBracket=rg2_mount_bracket_offset
  local gripperCoG=rg2_mount_cog_offset
  else:
  local gripperBracket=rg6_mount_bracket_offset
  local gripperCoG=rg6_mount_cog_offset
  end
  local gripperRotVec=rpy2rotvec([gripper_angle,0.0,0.0])
  local gripperMountOffset=p[0.0,0.0,gripperBracket,gripperRotVec[0],gripperRotVec[1],gripperRotVec[2]]
  local gripperCOGOffset=pose_trans(gripperMountOffset,gripperCoG)
  gripperCOGOffset=p[gripperCOGOffset[0],gripperCOGOffset[1],gripperCOGOffset[2],0.0,0.0,0.0]
  if ON_DEBUG_LOG:
  textmsg("RG Mount CoG command ended.")
  end
  return gripperCOGOffset
  end
  def rg_fcp_depth_calc_frame(tool_index=0):
  local gripperDepth=rg_Depth_arr[tool_index]
  local z_offset=-gripperDepth/1000.0
  return p[0.0,0.0,z_offset,0.0,0.0,0.0]
  end
  def rg_tcp_dynamic_get(tool_index=0):
  local offset=rg_fcp_depth_calc_frame(tool_index)
  return offset
  end
  def rg_payload_set(mass,tool_index=0,use_guard=False):
  if ON_DEBUG_LOG:
  textmsg("RG Payload mass command starting..")
  end
  if(tool_index==ON_DI_SECONDARY):
  local cogTool=[on_cog_workpiece_secondary[0],on_cog_workpiece_secondary[1],on_cog_workpiece_secondary[2]]
  else:
  local cogTool=[on_cog_workpiece_primary[0],on_cog_workpiece_primary[1],on_cog_workpiece_primary[2]]
  end
  if(use_guard and rg_Grip_detected_arr[tool_index]):
  local mass2set=mass
  rg_Grip_guard_arr[tool_index]=not on_ioqc
  else:
  local mass2set=0.0
  rg_Grip_guard_arr[tool_index]=False
  end
  on_payload_update_workpiece(mass2set,cogTool,tool_index)
  if ON_DEBUG_LOG:
  textmsg("RG Payload mass command ended.")
  end
  end

  #======    End of OnRobot RG TCP    ======#
  #======    OnRobot  Speedl    ======#

  on_speedl_thread_handler=0
  on_speedl_is_enabled=False
  on_speedl_is_running=False
  on_speedl_acc=0.0
  ft_speedl_hg_caranteen_reached=False
  ft_speedl_hg_caranteen_safemode=False
  on_speedl_for_ftcontrol=False
  on_speedl_for_move=False
  on_speedl_for_handguide=False
  on_speedl_for_insertpart=False
  on_speedl_for_depthcompensation=False
  on_speedl_for_center=False
  on_speedl_for_gecko=False
  on_speedl_acc=10000.0
  on_speedl_acc_to_zero=3.0
  ON_SPEEDL_FTCONTROL=1
  ON_SPEEDL_HANDGUIDE=2
  ON_SPEEDL_TRAJECTORY=3
  ON_SPEEDL_MOVE=ON_SPEEDL_TRAJECTORY
  ON_SPEEDL_INSERTPART=4
  ON_SPEEDL_DEPTHCOMP=5
  ON_SPEEDL_CENTER=6
  ON_SPEEDL_GECKO=7
  def on_wait_ms(time_ms):
  local sync_time=ceil(norm(time_ms/2.0))
  while(sync_time>0):
  sync_time=sync_time-1
  sync()
  end
  end
  def on_error(status_flag,message,title,stop_var=False):
  if(status_flag):
  popup(message,title=title,error=True,blocking=False)
  stop_var=True
  end
  return stop_var
  end
  def on_warning(status_flag,message,title,isPopupNeeded=False,is_shown=False):
  if(status_flag):
  if(not is_shown):
  if(isPopupNeeded):
  popup(message,title=title,warning=True,blocking=False)
  else:
  textmsg(title+": ",message)
  end
  is_shown=True
  end
  else:
  is_shown=False
  end
  return is_shown
  end
  def on_speedl_add_extra(speedBase,speedExtra):
  speedSum=ON_ZERO6D
  speedBaseP=p[speedBase[0],speedBase[1],speedBase[2],speedBase[3],speedBase[4],speedBase[5]]
  speedExtraP=p[speedExtra[0],speedExtra[1],speedExtra[2],speedExtra[3],speedExtra[4],speedExtra[5]]
  speedSumP=pose_add(speedExtraP,speedBaseP)
  speedSum=[speedSumP[0],speedSumP[1],speedSumP[2],speedSumP[3],speedSumP[4],speedSumP[5]]
  return speedSum
  end

  thread on_speedl_thread():
  if ON_DEBUG_LOG:
  textmsg("Speedl thread started..")
  end
  enter_critical
  on_speedl_is_running=True
  on_speedl_is_enabled=True
  exit_critical
  on_speedL=ON_ZERO6D
  on_speedL_last=ON_ZERO6D

  while on_speedl_is_running:
  on_speedBase=on_speedCB_get()
  on_speedL=on_speedBase


  if on_speedl_is_enabled:
  if(on_speedL==ON_ZERO6D):
  on_speedL=[on_speedL_last[0]/100,on_speedL_last[1]/100,on_speedL_last[2]/100,on_speedL_last[3]/100,on_speedL_last[4]/100,on_speedL_last[5]/100]
  end
  speedl(on_speedL,a=on_speedl_acc,t=speedlTime)
  else:
  speedl(ON_ZERO6D,a=on_speedl_acc_to_zero,t=speedlTime)
  end
  on_speedL_last=on_speedL
  end

  on_speedL=ON_ZERO6D
  if ON_DEBUG_LOG:
  textmsg("Speedl thread ended.")
  end
  end
  def on_speedl_integer_get():
  local speedl_integer=binary_list_to_integer([on_speedl_for_ftcontrol,on_speedl_for_handguide,on_speedl_for_move,on_speedl_for_insertpart,on_speedl_for_depthcompensation,on_speedl_for_center,on_speedl_for_gecko])
  return speedl_integer
  end
  def on_speedl_start_for(speedl_id):
  if(speedl_id==ON_SPEEDL_FTCONTROL):
  on_speedl_for_ftcontrol=True
  elif(speedl_id==ON_SPEEDL_HANDGUIDE):
  on_speedl_for_handguide=True
  elif(speedl_id==ON_SPEEDL_TRAJECTORY):
  on_speedl_for_move=True
  elif(speedl_id==ON_SPEEDL_INSERTPART):
  on_speedl_for_insertpart=True
  elif(speedl_id==ON_SPEEDL_DEPTHCOMP):
  on_speedl_for_depthcompensation=True
  elif(speedl_id==ON_SPEEDL_CENTER):
  on_speedl_for_center=True
  elif(speedl_id==ON_SPEEDL_GECKO):
  on_speedl_for_gecko=True
  else:
  textmsg("Unknown Start speedl ID received: ",speedl_id)
  end
  local speedl_integer=on_speedl_integer_get()
  if not(speedl_integer==0):
  if not on_speedl_is_running:
  on_speedl_thread_handler=run on_speedl_thread()
  end
  end
  return on_speedl_is_running
  end
  def on_speedl_stop_for(speedl_id,brake=10,brakeRot=10):
  if(speedl_id==ON_SPEEDL_FTCONTROL):
  on_speedl_for_ftcontrol=False
  elif(speedl_id==ON_SPEEDL_HANDGUIDE):
  on_speedl_for_handguide=False
  elif(speedl_id==ON_SPEEDL_TRAJECTORY):
  on_speedl_for_move=False
  elif(speedl_id==ON_SPEEDL_INSERTPART):
  on_speedl_for_insertpart=False
  elif(speedl_id==ON_SPEEDL_DEPTHCOMP):
  on_speedl_for_depthcompensation=False
  elif(speedl_id==ON_SPEEDL_CENTER):
  on_speedl_for_center=False
  elif(speedl_id==ON_SPEEDL_GECKO):
  on_speedl_for_gecko=False
  on_speedGecko_set(ON_ZERO6D)
  else:
  textmsg("Unknown Stop speedl ID received: ",speedl_id)
  end
  local speedl_integer=on_speedl_integer_get()
  if(speedl_integer==0):
  if(on_speedl_is_running):
  kill on_speedl_thread_handler
  enter_critical
  on_speedl_is_running=False
  exit_critical

  end
  if ON_DEBUG_LOG:
  textmsg("Speedl thread stopped")
  end
  stopl(brake,brakeRot)
  end
  return on_speedl_is_running
  end
  def on_speedl_pause():
  on_speedl_is_enabled=False
  return on_speedl_integer_get()
  end
  def on_speedl_resume():
  on_speedl_is_enabled=True
  return on_speedl_integer_get()
  end

  #======    End of OnRobot  Speedl    ======#
  #======    OnRobot RG Engine Messages    ======#

  rg_error_title="OnRobot - RG error"
  rg_device_id_waiting="Waiting for valid OnRobot RG ID..."
  rg_device_id_timeout="Waiting for valid OnRobot RG ID timed out.<br>Program halted."
  rg_data_error_title="OnRobot - RG Data error"
  rg_data_error_type="No or unknown Gripper connected."
  rg_data_warning_title="OnRobot - RG Data warning:"
  rg_status_error_title="OnRobot - RG Status error"
  rg_status_error_missing="Communication problem with an RG gripper. Please check the device.<br>Program halted."
  rg_else_error="Unknown error code:"
  rg_status_msg_single="RG status:"
  rg_data_error_bit0_single="Wrong size of float data received."
  rg_data_error_bit1_single="Wrong size of integer data received."
  rg_data_error_bit2_single="Wrong size of boolean data received."
  rg_status_error_mismatch_single="The RG's Status is not matching with its Safety Switches' state."
  rg_status_error_s1_triggered_single="The S1 Safety Switch has been triggered.<br>Please restart the RG gripper."
  rg_status_error_s1_pushed_single="The S1 Safety Switch has been pushed."
  rg_status_error_s2_triggered_single="The S2 Safety Switch has been triggered.<br>Please restart the RG gripper."
  rg_status_error_s2_pushed_single="The S2 Safety Switch has been pushed."
  rg_status_error_safety_system_single="Safety System error occured.<br>Please restart the RG gripper."
  rg_status_msg_primary="RG Primary status:"
  rg_data_error_bit0_primary="Wrong size of float data received for Primary RG."
  rg_data_error_bit1_primary="Wrong size of integer data received for Primary RG."
  rg_data_error_bit2_primary="Wrong size of boolean data received for Primary RG."
  rg_status_error_mismatch_primary="The Primary RG's Status is not matching with its Safety Switches' state."
  rg_status_error_s1_pushed_primary="The S1 Safety Switch has been pushed on Primary RG."
  rg_status_error_s1_triggered_primary="The S1 Safety Switch has been triggered on Primary RG.<br>Please restart the Primary RG gripper."
  rg_status_error_s2_pushed_primary="The S2 Safety Switch has been pushed on Primary RG."
  rg_status_error_s2_triggered_primary="The S2 Safety Switch has been triggered on Primary RG.<br>Please restart the Primary RG gripper."
  rg_status_error_safety_system_primary="Safety System error occured.<br>Please restart the Primary RG gripper."
  rg_status_msg_secondary="RG Secondary status:"
  rg_data_error_bit0_secondary="Wrong size of float data received for Secondary RG."
  rg_data_error_bit1_secondary="Wrong size of integer data received for Secondary RG."
  rg_data_error_bit2_secondary="Wrong size of boolean data received for Secondary RG."
  rg_status_error_mismatch_secondary="The Secondary RG's Status is not matching with its Safety Switches' state."
  rg_status_error_s1_pushed_secondary="The S1 Safety Switch has been pushed on Secondary RG."
  rg_status_error_s1_triggered_secondary="The S1 Safety Switch has been triggered on Secondary RG.<br>Please restart the Secondary RG gripper."
  rg_status_error_s2_pushed_secondary="The S2 Safety Switch has been pushed on Secondary RG."
  rg_status_error_s2_triggered_secondary="The S2 Safety Switch has been triggered on Secondary RG.<br>Please restart the Secondary RG gripper."
  rg_status_error_safety_system_secondary="The Safety System error.<br>Please restart the Secondary RG gripper."

  #======    End of OnRobot RG Engine Messages    ======#
  #======    OnRobot RG Engine    ======#

  rg_dataProcess_running=False
  rg_start_flange=ON_ZEROPOSE
  rg_start_pose=ON_ZEROPOSE
  RG_STATUS_IGNORE_SHIFT=4
  def rg_status_int_get(tool_index):
  local status_int=binary_list_to_integer([rg_S1_pushed_arr[tool_index],rg_S1_triggered_arr[tool_index],rg_S2_pushed_arr[tool_index],rg_S2_triggered_arr[tool_index],rg_Safety_error_arr[tool_index]])
  return status_int
  end
  def rg_dataProcess_status_errors(rg_stop=False):
  enter_critical
  local tool_index=rg_index
  if(tool_index==ON_DI_DUAL):
  tool_index=ON_DI_SECONDARY
  rg_stop=on_error((rg_device_id_arr[tool_index]!=tool_index),rg_status_error_missing,rg_status_error_title,rg_stop)
  rg_stop=on_error((rg_product_code_arr[tool_index]==ON_DEVICE_ID_MISSING),rg_status_error_missing,rg_status_error_title,rg_stop)
  tool_index=ON_DI_PRIMARY
  end
  rg_stop=on_error((rg_device_id_arr[tool_index]!=tool_index),rg_status_error_missing,rg_status_error_title,rg_stop)
  rg_stop=on_error((rg_product_code_arr[tool_index]==ON_DEVICE_ID_MISSING),rg_status_error_missing,rg_status_error_title,rg_stop)

  local switch_error_single=rg_status_int_get(tool_index)
  local status_error_single=floor(rg_Status_arr[tool_index]/RG_STATUS_IGNORE_SHIFT)
  if(status_error_single!=switch_error_single):
  on_warning(((status_error_single-switch_error_single)>0),str_cat(rg_else_error,rg_Status_arr[tool_index]),rg_status_error_title)
  end
  if(switch_error_single!=0):
  rg_stop=on_error(rg_S1_pushed_arr[tool_index],rg_status_error_s1_pushed_single,rg_status_error_title,rg_stop)
  rg_stop=on_error(rg_S1_triggered_arr[tool_index],rg_status_error_s1_triggered_single,rg_status_error_title,rg_stop)
  rg_stop=on_error(rg_S2_pushed_arr[tool_index],rg_status_error_s2_pushed_single,rg_status_error_title,rg_stop)
  rg_stop=on_error(rg_S2_triggered_arr[tool_index],rg_status_error_s2_triggered_single,rg_status_error_title,rg_stop)
  rg_stop=on_error(rg_Safety_error_arr[tool_index],rg_status_error_safety_system_single,rg_status_error_title,rg_stop)
  end

  exit_critical
  return rg_stop
  end
  def rg_dataProcess():
  enter_critical
  local tool_index=rg_index
  if tool_index==ON_DI_DUAL:
  rg_Width_primary=rg_Width_arr[ON_DI_PRIMARY]
  rg_Depth_primary=rg_Depth_arr[ON_DI_PRIMARY]
  rg_DepthRel_primary=rg_DepthRel_arr[ON_DI_PRIMARY]
  rg_Busy_primary=rg_Busy_arr[ON_DI_PRIMARY]
  rg_Grip_detected_primary=rg_Grip_detected_arr[ON_DI_PRIMARY]
  rg_Width_secondary=rg_Width_arr[ON_DI_SECONDARY]
  rg_Depth_secondary=rg_Depth_arr[ON_DI_SECONDARY]
  rg_DepthRel_secondary=rg_DepthRel_arr[ON_DI_SECONDARY]
  rg_Busy_secondary=rg_Busy_arr[ON_DI_SECONDARY]
  rg_Grip_detected_secondary=rg_Grip_detected_arr[ON_DI_SECONDARY]
  else:
  rg_Width=rg_Width_arr[tool_index]
  rg_Depth=rg_Depth_arr[tool_index]
  rg_DepthRel=rg_DepthRel_arr[tool_index]
  rg_Busy=rg_Busy_arr[tool_index]
  rg_Grip_detected=rg_Grip_detected_arr[tool_index]
  end
  exit_critical
  end
  thread rg_dataProcess_thread():
  if ON_DEBUG_LOG:
  textmsg("Starting rg_dataProcess thread")
  end
  while rg_dataProcess_running:
  sync()
  local rg_stop=False
  rg_stop=rg_dataProcess_status_errors(rg_stop)
  if rg_stop:
  halt
  end
  rg_dataProcess()
  end
  if ON_DEBUG_LOG:
  textmsg("Stopping rg_dataProcess thread")
  end
  end
  def rg_index_get():
  return rg_index
  end

  #======    End of OnRobot RG Engine    ======#
  rg_mounting_angle_arr[0] = 0.0
  rg_fingertip_arr[0] = 4.599999904632568
  rg_Depth_arr[0] = 4.599999904632568
  textmsg(on_devices_primary_log, ": Quick Changer + RG2 + [0.0, 0.0, 0.0, 0.0, 0.0, 0.0]")
  on_follow_tcp = False
  on_tcp_active_is_primary = True
  on_tcp_adapters_array = []
  on_cog_adapters_array = []
  on_mass_adapters_array = []
  on_tcp_qc_primary = p[0.0, 0.0, 0.0136, 0.0, 0.0, 0.0]
  on_cog_qc_primary = p[0.0, 0.0, 0.004, 0.0, 0.0, 0.0]
  on_mass_qc_primary = 0.06
  on_tcp_gripper_static_primary = rg_mount_tcp(rg_mounting_angle_arr[0])
  on_cog_gripper_primary = rg_mount_cog(rg_mounting_angle_arr[0])
  on_mass_gripper_primary = 0.78
  on_tcp_workpiece_primary = p[0.0, 0.0, 0.0, 0.0, 0.0, 0.0]
  on_cog_workpiece_primary = p[0.0, 0.0, 0.0, 0.0, 0.0, 0.0]
  on_mass_workpiece_primary = 0.0

  #======    End of OnRobot RG Depth    ======#
  #======    OnRobot RG Width Messages    ======#

  rg_grip_title="OnRobot - RG Grip"
  rg_grip_return_error_n1="RG Grip command returned with error.<br>Please be sure that the required width is between the limits.<br>Program halted."

  #======    End of OnRobot RG Width Messages    ======#
  #======    OnRobot RG Width    ======#

  RG_MIN_WIDTH=0
  RG_MAX_WIDTH_RG2=110
  RG_MAX_WIDTH_RG6=160
  RG_MIN_FORCE=0
  RG_MAX_FORCE_RG2=40
  RG_MAX_FORCE_RG6=120
  rg__grip_param_warning_width="The parameter 'width' is out of the limits. Limited value sent: "
  rg__grip_param_warning_force="The parameter 'force' is out of the limits. Limited value sent: "
  def rg_depth_compensate(tool_index,start_depth_mm):
  local timeout=0
  while not rg_Busy_arr[tool_index]:
  sleep(0.008)
  timeout=timeout+1
  if timeout>20:
  break
  end
  end
  local start_pose=get_forward_kin()
  if(tool_index==ON_DI_SECONDARY):
  local tcp_static=on_tcp_static_secondary
  else:
  local tcp_static=on_tcp_static_primary
  end
  local t_w_rg=pose_trans(get_actual_tool_flange_pose(),tcp_static)
  local t_rg_w=pose_inv(t_w_rg)
  local compensation_depth_mm=0
  local after_ready_continue_count=10
  while True:
  local busy=rg_Busy_arr[tool_index]
  if not busy:
  if after_ready_continue_count>0:
  after_ready_continue_count=after_ready_continue_count-1
  else:
  break
  end
  end
  local measure_depth_mm=rg_Depth_arr[tool_index]
  compensation_depth_mm=measure_depth_mm-start_depth_mm
  local target_pose=pose_add(start_pose,pose_trans(pose_trans(t_w_rg,p[0,0,compensation_depth_mm/1000.0,0,0,0]),t_rg_w))
  servoj(get_inverse_kin(target_pose),t=0.008,lookahead_time=0.033,gain=1500)
  end
  stopj(20)
  end
  def rg_grip(width,force,tool_index=0,blocking=True,depth_comp=False,popupmsg=True):
  if ON_DEBUG_LOG:
  textmsg("RG Grip start..")
  end
  local retVal=0
  local limitOffset=(2.0*rg_fingertip_arr[tool_index])
  local width2send=width
  if limitOffset>0:
  local minWidth=RG_MIN_WIDTH
  else:
  local minWidth=RG_MIN_WIDTH-limitOffset
  end
  if not(width2send>=minWidth):
  width2send=minWidth
  textmsg(rg__grip_param_warning_width,width2send)
  elif not(force>=RG_MIN_FORCE):
  force=RG_MIN_FORCE
  textmsg(rg__grip_param_warning_force,force)
  end
  if(rg_product_code_arr[tool_index]==RG_DEVICE_ID_RG6):
  if not(width2send<=RG_MAX_WIDTH_RG6-limitOffset):
  width2send=RG_MAX_WIDTH_RG6-limitOffset
  textmsg(rg__grip_param_warning_width,width2send)
  elif not(force<=RG_MAX_FORCE_RG6):
  force=RG_MAX_FORCE_RG6
  textmsg(rg__grip_param_warning_force,force)
  end
  else:
  if not(width2send<=RG_MAX_WIDTH_RG2-limitOffset):
  width2send=RG_MAX_WIDTH_RG2-limitOffset
  textmsg(rg__grip_param_warning_width,width2send)
  elif not((force<=RG_MAX_FORCE_RG2)):
  force=RG_MAX_FORCE_RG2
  textmsg(rg__grip_param_warning_force,force)
  end
  end
  rg_Grip_guard_arr[tool_index]=False
  sync()
  if(tool_index==ON_DI_SECONDARY):
  local isPrimary=False
  else:
  local isPrimary=True
  end
  if(on_follow_tcp):
  on_tcp_set_actual_to(isPrimary)
  end
  if depth_comp:
  local start_depth_mm=rg_Depth_arr[tool_index]
  end
  sync()
  retVal=on_tool_xmlrpc.rg_grip(tool_index,width2send+0.0,force+0.0)
  if(retVal!=0):
  popup(rg_grip_return_error_n1,rg_grip_title,error=True,blocking=False)
  halt
  end
  if depth_comp:
  rg_depth_compensate(tool_index,start_depth_mm)
  end
  if blocking:
  if not depth_comp:
  local timeout=0
  while not rg_Busy_arr[tool_index]:
  sleep(0.008)
  timeout=timeout+1
  if timeout>20:
  break
  end
  end
  end
  while(rg_Busy_arr[tool_index]==True):
  sync()
  end
  end
  if(on_follow_tcp):
  on_tcp_update(isPrimary)
  end
  if ON_DEBUG_LOG:
  textmsg("RG Grip ended.")
  end
  return retVal
  end

  #======    End of OnRobot RG Width    ======#
  #======    OnRobot VG Monitor Messages    ======#

  rg_monitor_error_title="OnRobot - RG Grip lost"
  rg_monitor_grip_lost_error="Grip lost detected.<br>Program halted."

  #======    End of OnRobot VG Monitor Messages    ======#
  #======    OnRobot RG Monitor    ======#

  thread rg_monitor_thread():
  while True:
  sync()
  local rg_error=False
  if(rg_index==ON_DI_DUAL):
  local tool_index=ON_DI_SECONDARY
  rg_error=rg_monitor_check(tool_index)
  local tool_index=ON_DI_PRIMARY
  else:
  local tool_index=rg_index
  end
  rg_error=rg_error or rg_monitor_check(tool_index)
  if rg_error:
  halt
  end
  end
  end
  def rg_monitor_check(tool_index=0):
  local error=False
  if rg_Grip_guard_arr[tool_index]and not rg_Grip_detected_arr[tool_index]:
  popup(rg_monitor_grip_lost_error,title=rg_monitor_error_title,error=True,blocking=False)
  rg_payload_set(0,tool_index=tool_index)
  error=True
  end
  return error
  end

  #======    End of OnRobot RG Monitor    ======#
  #======    OnRobot Run    ======#

  on_portopen_javaSocket()
  sync()
  textmsg(on_xmlrpc_start_ip,on_conn_ip)
  if(ON_REG_USE_TOOL):
  on_regStart_conn=[ON_CONN_SHIFT_BOOL,ON_CONN_SHIFT_INT,ON_CONN_SHIFT_FLOAT]
  on_regSum_conn=[ON_CONN_REG_SUM_BOOL,ON_CONN_REG_SUM_INT,ON_CONN_REG_SUM_FLOAT]
  on_rtde_feed_open(on_conn_ip,on_conn_rtde_feed_name,on_regStart_conn,on_regSum_conn,ON_REGISTERS_SPEEDL_FLOAT)
  sync()
  textmsg(on_xmlrpc_start_ip,on_tool_ip)
  on_regStart_tool=[ON_TOOL_SHIFT_BOOL,ON_TOOL_SHIFT_INT,ON_TOOL_SHIFT_FLOAT]
  on_regSum_tool=[ON_TOOL_REG_SUM_BOOL,ON_TOOL_REG_SUM_INT,ON_TOOL_REG_SUM_FLOAT]
  on_rtde_feed_open(on_tool_ip,on_tool_rtde_feed_name,on_regStart_tool,on_regSum_tool,0)
  sync()
  else:
  on_regStart_conn=[ON_CONN_SHIFT_BOOL,ON_CONN_SHIFT_INT,ON_CONN_SHIFT_FLOAT]
  on_regSum_conn=[ON_CONN_REG_SUM_BOOL,ON_CONN_REG_SUM_INT,ON_CONN_REG_SUM_FLOAT]
  on_rtde_feed_open(on_conn_ip,on_conn_rtde_feed_name,on_regStart_conn,on_regSum_conn,ON_REGISTERS_SPEEDL_FLOAT)
  sync()
  end
  on_set_rtde_watchdog(updateHz=0.2)
  sync()
  on_dataProcess_thrd=run on_dataProcess_thread()
  sync()
  on_tcp_init_adapters()
  on_payload_init_adapters()
  on_tcp_init_primary()
  on_payload_init_primary()

  on_tcp_update_custom()
  on_tcp_set_actual_to(on_tcp_active_is_primary)
  if(on_follow_tcp):
  on_payload_set_actual()
  end
  on_watchdog_thrd=run on_set_watchdog_thread()
  sync()
  def done_waiting_for_init(device_name,product_code,tool_index=0):
  textmsg(str_cat(device_name,str_cat(str_cat("[",tool_index),"]: ")),product_code)
  end

  #======    End of OnRobot Run    ======#
  #======    OnRobot QC Start    ======#

  if(on_toolConnector):
  tc_setup_tool()
  end
  sync()

  #======    End of OnRobot QC Start    ======#
  #======    OnRobot RG Run    ======#

  def rg_wait_for_init(tool_index):
  local rg_timeout=0
  while not((rg_product_code_arr[tool_index]==RG_DEVICE_ID_RG2)or(rg_product_code_arr[tool_index]==RG_DEVICE_ID_RG6)):
  sync()
  rg_timeout=rg_timeout+1
  if(rg_timeout>ON_INIT_TIMEOUT):
  popup(rg_device_id_timeout,rg_error_title,error=True,blocking=False)
  halt
  end
  end
  done_waiting_for_init("RG",rg_product_code_arr[tool_index],tool_index)
  end
  rg_dataRead_running=True
  sync()
  rg_dataRead_thrd=run rg_dataRead_thread()
  sync()
  textmsg(rg_device_id_waiting)
  if(rg_index==ON_DI_DUAL):
  rg_wait_for_init(ON_DI_PRIMARY)
  rg_wait_for_init(ON_DI_SECONDARY)
  else:
  rg_wait_for_init(rg_index)
  end
  sync()
  rg_dataProcess_running=True
  sync()
  rg_dataProcess_thrd=run rg_dataProcess_thread()
  sync()
  rg_monitor_thread_handle=run rg_monitor_thread()
  sync()

  #======    End of OnRobot RG Run    ======#
  # end: URCap Installation Node
  global home_p=p[.359452291236, .012314525122, .397104007426, 2.228474804439, -2.207095578885, -.005864977278]
  global home_q=[0.5392290949821472, -1.4658818331411858, -2.184360980987549, -4.210199495355123, -1.5756142775165003, -2.6091490427600306]
  global Waypoint_1_p=p[.421489587850, -.013304754036, .395906972318, 2.228579159892, -2.206885102157, -.005749914791]
  global Waypoint_1_q=[0.39398816227912903, -1.5834981403746546, -2.075856924057007, -4.2014082870879115, -1.5745413939105433, -2.754477087651388]
  global Waypoint_3_p=p[.421478074770, -.013324872178, .274291336021, 2.228531548836, -2.206952746442, -.005794124343]
  global Waypoint_3_q=[0.39406681060791016, -1.7239324055113734, -2.1863694190979004, -3.95045866588735, -1.5742085615741175, -2.7536607424365442]
  global Waypoint_2_p=p[.180759056879, -.218870541575, .390032721103, 2.228497220874, -2.207079648930, -.005641311239]
  global Waypoint_2_q=[-0.2180421988116663, -1.3045593363097687, -2.32352614402771, -4.232248922387594, -1.5709827581988733, -3.36653715768923]
  global Waypoint_4_p=p[.180762311825, -.218865707852, .274724104396, 2.228550080175, -2.207124147127, -.005632451855]
  global Waypoint_4_q=[-0.21767074266542608, -1.4666959282806893, -2.4519081115722656, -3.9416915378966273, -1.570637051259176, -3.3653391043292444]
  global Waypoint_5_p=p[.180742544246, -.218864877734, .386037734354, 2.228494552468, -2.207187456003, -.005679767184]
  global Waypoint_5_q=[-0.21805936494936162, -1.3087391716292878, -2.3285937309265137, -4.222982545892233, -1.57104999223818, -3.366477076207296]
  global above2_p=p[.415149015504, .046900275077, .386038228830, 2.228486790383, -2.207167316029, -.005679434851]
  global above2_q=[0.5420307517051697, -1.585785528222555, -2.093414783477783, -4.181149622003073, -1.575416390095846, -2.6062117258654993]
  global appr_2_p=p[.424025119840, .036453055985, .276202945805, 2.228421507966, -2.207205276843, -.005750959906]
  global appr_2_q=[0.5070622563362122, -1.7273971043028773, -2.1773815155029297, -3.9556778870024623, -1.5749056974994105, -2.6405168215381067]
  global Waypoint_6_p=p[.424033285965, .036490434353, .346540172866, 2.228551980283, -2.207053599322, -.005679311005]
  global Waypoint_6_q=[0.5070841312408447, -1.6402880154051722, -2.118475914001465, -4.101694246331686, -1.5750930945025843, -2.641012970601217]
  global above_des2_p=p[.218752662814, -.219185090783, .348476289511, 2.228788233078, -2.206998434932, -.005614183283]
  global above_des2_q=[-0.1874788443194788, -1.4139403116754075, -2.327842950820923, -4.118523975411886, -1.5711100737201136, -3.335789982472555]
  global Waypoint_7_p=p[.218739875303, -.219198786131, .279670710543, 2.228713454329, -2.207113400969, -.005610223887]
  global Waypoint_7_q=[-0.18737680116762334, -1.5149477657726784, -2.3973138332366943, -3.948029418984884, -1.570864502583639, -3.335127655659811]
  global above_start3_p=p[.476970296740, -.013897699301, .361840783109, 2.228757880509, -2.207061217753, -.005565328800]
  global above_start3_q=[0.3443509638309479, -1.7101017437376917, -2.0068917274475098, -4.143554349938864, -1.5740874449359339, -2.8039372603045862]
  global pick3_p=p[.476970272495, -.013876044234, .277290954381, 2.228790479633, -2.207044965651, -.005617930906]
  global pick3_q=[0.34444117546081543, -1.804579874078268, -2.0756688117980957, -3.980302473107809, -1.57387620607485, -2.803432289754049]
  global Waypoint_8_p=p[.256105412964, -.218931053662, .372722929963, 2.228789403332, -2.207012661408, -.005586442423]
  global Waypoint_8_q=[-0.16279346147646123, -1.4442329865745087, -2.2523810863494873, -4.163722654382223, -1.5712655226336878, -3.3112130800830286]
  global Waypoint_9_p=p[.256107606788, -.218931520606, .280483573827, 2.228754436535, -2.206992067667, -.005629886323]
  global Waypoint_9_q=[-0.16260224977602178, -1.5681753319552918, -2.3444364070892334, -3.9477721653380335, -1.5709260145770472, -3.3104143778430384]
  global above4_p=p[.475180432478, .034611087756, .374297722738, -2.240969228761, 2.201709247231, -.000043439770]
  global above4_q=[0.44707125425338745, -1.6951524219908656, -1.9970643520355225, -4.162305732766622, -1.5730255285846155, -2.7091599146472376]
  global Waypoint_10_p=p[.475185199327, .034616319337, .276924349654, 2.240934996990, -2.201661965571, -.000007202828]
  global Waypoint_10_q=[0.4471415877342224, -1.802054067651266, -2.0782227516174316, -3.9743522606291712, -1.5727418104754847, -2.7085915247546595]
  global Waypoint_11_p=p[.291878079444, -.217433283291, .358649983572, -2.240985552805, 2.201719537788, -.000110616791]
  global Waypoint_11_q=[-0.14086753526796514, -1.5126863953522225, -2.219794750213623, -4.1220125160613, -1.573118034993307, -3.297021452580587]
  global Waypoint_12_p=p[.291891548237, -.217428284089, .281086670334, 2.240975321956, -2.201700743893, .000109023186]
  global Waypoint_12_q=[-0.14071542421449834, -1.6152249775328578, -2.2927207946777344, -3.9465648136534632, -1.5728204886065882, -3.2963934580432337]
  while (True):
    $ 1 "Robot Program"
    $ 2 "MoveL"
    $ 3 "home" "breakAfter"
    movel(home_p, a=1.2, v=0.25)
    # begin: URCap Program Node
    #   Source: OnRobot, 6.2.0, OnRobot A/S
    #   Type: RG Grip
    $ 4 "RG Grip"
on_return = rg_grip(40.0, 3.0, tool_index = 0, blocking = True, depth_comp = False, popupmsg = True)
rg_payload_set(mass = 0.0, tool_index = 0, use_guard = True)
    # end: URCap Program Node
    $ 5 "Waypoint_1" "breakAfter"
    movel(Waypoint_1_p, a=1.2, v=0.25)
    $ 6 "Waypoint_3" "breakAfter"
    movel(Waypoint_3_p, a=1.2, v=0.25)
    # begin: URCap Program Node
    #   Source: OnRobot, 6.2.0, OnRobot A/S
    #   Type: RG Grip
    $ 7 "RG Grip"
on_return = rg_grip(32.0, 3.0, tool_index = 0, blocking = True, depth_comp = False, popupmsg = True)
rg_payload_set(mass = 0.0, tool_index = 0, use_guard = True)
    # end: URCap Program Node
    $ 8 "Waypoint_1" "breakAfter"
    movel(Waypoint_1_p, a=1.2, v=0.25)
    $ 9 "MoveL"
    $ 10 "Waypoint_2" "breakAfter"
    movel(Waypoint_2_p, a=1.2, v=0.25)
    $ 11 "Waypoint_4" "breakAfter"
    movel(Waypoint_4_p, a=1.2, v=0.25)
    # begin: URCap Program Node
    #   Source: OnRobot, 6.2.0, OnRobot A/S
    #   Type: RG Grip
    $ 12 "RG Grip"
on_return = rg_grip(40.0, 3.0, tool_index = 0, blocking = True, depth_comp = False, popupmsg = True)
rg_payload_set(mass = 0.0, tool_index = 0, use_guard = True)
    # end: URCap Program Node
    $ 13 "Waypoint_5" "breakAfter"
    movel(Waypoint_5_p, a=1.2, v=0.25)
    $ 14 "above2" "breakAfter"
    movel(above2_p, a=1.2, v=0.25)
    $ 15 "appr_2" "breakAfter"
    movel(appr_2_p, a=1.2, v=0.25)
    # begin: URCap Program Node
    #   Source: OnRobot, 6.2.0, OnRobot A/S
    #   Type: RG Grip
    $ 16 "RG Grip"
on_return = rg_grip(32.0, 3.0, tool_index = 0, blocking = True, depth_comp = True, popupmsg = True)
rg_payload_set(mass = 0.0, tool_index = 0, use_guard = True)
    # end: URCap Program Node
    $ 17 "Waypoint_6" "breakAfter"
    movel(Waypoint_6_p, a=1.2, v=0.25)
    $ 18 "above_des2" "breakAfter"
    movel(above_des2_p, a=1.2, v=0.25)
    $ 19 "Waypoint_7" "breakAfter"
    movel(Waypoint_7_p, a=1.2, v=0.25)
    # begin: URCap Program Node
    #   Source: OnRobot, 6.2.0, OnRobot A/S
    #   Type: RG Grip
    $ 20 "RG Grip"
on_return = rg_grip(40.0, 3.0, tool_index = 0, blocking = True, depth_comp = False, popupmsg = True)
rg_payload_set(mass = 0.0, tool_index = 0, use_guard = True)
    # end: URCap Program Node
    $ 21 "above_des2" "breakAfter"
    movel(above_des2_p, a=1.2, v=0.25)
    $ 22 "MoveL"
    $ 23 "above_start3" "breakAfter"
    movel(above_start3_p, a=1.2, v=0.25)
    $ 24 "pick3" "breakAfter"
    movel(pick3_p, a=1.2, v=0.25)
    # begin: URCap Program Node
    #   Source: OnRobot, 6.2.0, OnRobot A/S
    #   Type: RG Grip
    $ 25 "RG Grip"
on_return = rg_grip(32.0, 3.0, tool_index = 0, blocking = True, depth_comp = True, popupmsg = True)
rg_payload_set(mass = 0.0, tool_index = 0, use_guard = True)
    # end: URCap Program Node
    $ 26 "above_start3" "breakAfter"
    movel(above_start3_p, a=1.2, v=0.25)
    $ 27 "Waypoint_8" "breakAfter"
    movel(Waypoint_8_p, a=1.2, v=0.25)
    $ 28 "Waypoint_9" "breakAfter"
    movel(Waypoint_9_p, a=1.2, v=0.25)
    # begin: URCap Program Node
    #   Source: OnRobot, 6.2.0, OnRobot A/S
    #   Type: RG Grip
    $ 29 "RG Grip"
on_return = rg_grip(40.0, 3.0, tool_index = 0, blocking = True, depth_comp = False, popupmsg = True)
rg_payload_set(mass = 0.0, tool_index = 0, use_guard = True)
    # end: URCap Program Node
    $ 30 "Waypoint_8" "breakAfter"
    movel(Waypoint_8_p, a=1.2, v=0.25)
    $ 31 "MoveL"
    $ 32 "above4" "breakAfter"
    movel(above4_p, a=1.2, v=0.25)
    $ 33 "Waypoint_10" "breakAfter"
    movel(Waypoint_10_p, a=1.2, v=0.25)
    # begin: URCap Program Node
    #   Source: OnRobot, 6.2.0, OnRobot A/S
    #   Type: RG Grip
    $ 34 "RG Grip"
on_return = rg_grip(32.0, 3.0, tool_index = 0, blocking = True, depth_comp = True, popupmsg = True)
rg_payload_set(mass = 0.0, tool_index = 0, use_guard = True)
    # end: URCap Program Node
    $ 35 "above4" "breakAfter"
    movel(above4_p, a=1.2, v=0.25)
    $ 36 "Waypoint_11" "breakAfter"
    movel(Waypoint_11_p, a=1.2, v=0.25)
    $ 37 "Waypoint_12" "breakAfter"
    movel(Waypoint_12_p, a=1.2, v=0.25)
    # begin: URCap Program Node
    #   Source: OnRobot, 6.2.0, OnRobot A/S
    #   Type: RG Grip
    $ 38 "RG Grip"
on_return = rg_grip(40.0, 3.0, tool_index = 0, blocking = True, depth_comp = False, popupmsg = True)
rg_payload_set(mass = 0.0, tool_index = 0, use_guard = True)
    # end: URCap Program Node
    $ 39 "Waypoint_11" "breakAfter"
    movel(Waypoint_11_p, a=1.2, v=0.25)
    $ 40 "MoveJ"
    $ 41 "home" "breakAfter"
    movej(get_inverse_kin(home_p, qnear=home_q), a=1.3962634015954636, v=1.0471975511965976)
    $ 42 "Halt"
    halt
  end
end
